FUNCTION_BLOCK FB_EVENT_LOGGER IMPLEMENTS I_EVENT_LOGGER
VAR
  fbAlarm:                        FB_TcAlarm;
  fbMessage:                      FB_TcMessage;
  bError:                         BOOL;
  bInfo:                          BOOL;
  bWarning:                       BOOL;
  uiSeq:                          ARRAY [1..3] OF UINT := [0, 0, 0];
  udiID:                          UDINT;
	sMsg:                           T_MaxString;
  bWithConfirmation:              BOOL;
END_VAR

IF bInfo THEN
  CASE uiSeq[1] OF
    0:
      fbMessage.CreateEx(TC_EVENTS.Info.IndividualInfoMsg, 0);
      uiSeq[1] := 1;
    1:
      fbMessage.ipArguments.Clear().AddDInt(udiID).AddString(sMsg);
      fbMessage.Send(0);
      uiSeq[1] := 2;
    2:
      bInfo := FALSE;
      uiSeq[1] := 0;
	END_CASE
END_IF

IF bWarning THEN
  CASE uiSeq[2] OF
    0:
      fbMessage.CreateEx(TC_EVENTS.Warnings.IndividualWarningMsg, 0);
      uiSeq[2] := 1;
    1:
      fbMessage.ipArguments.Clear().AddDInt(udiID).AddString(sMsg);
      fbMessage.Send(0);
      uiSeq[2] := 2;
    2:
      bWarning := FALSE;
      uiSeq[2] := 0;
	END_CASE
END_IF

IF bError THEN
  CASE uiSeq[3] OF
    0:
      fbAlarm.CreateEx(TC_EVENTS.Errors.IndividualErrMsg, bWithConfirmation, 0);
      uiSeq[3] := 1;
    1:
      fbAlarm.ipArguments.Clear().AddDInt(udiID).AddString(sMsg);
      fbAlarm.Raise(0);
      uiSeq[3] := 2;
    2:
      bError := FALSE;
      uiSeq[3] := 0;
	END_CASE
END_IF

METHOD M_ErrorMsg : BOOL
VAR_INPUT
	udiID:                        UDINT;
	sMsg:                         T_MaxString;
  bWithConfirmation:            BOOL;
END_VAR
M_ErrorMsg := THIS^.uiSeq[3] = 2;

// Assign input
THIS^.udiID := udiID;
THIS^.sMsg := sMsg;
THIS^.bWithConfirmation := bWithConfirmation;

THIS^.bError := TRUE;
END_METHOD

METHOD M_InfoMsg : BOOL
VAR_INPUT
	udiID	: UDINT;
	sMsg	: Tc2_System.T_MaxString;
END_VAR
M_InfoMsg := THIS^.uiSeq[1] = 2;

// Assign input
THIS^.udiID := udiID;
THIS^.sMsg := sMsg;

THIS^.bInfo := TRUE;
END_METHOD

{warning 'Methodenimplementierung hinzufügen'}
(*=== Method: M_Run  ============================================

 @brief: Here is the global code (Timer, Event, Flange,...)*)
METHOD M_Run
END_METHOD

METHOD M_WarningMsg : BOOL
VAR_INPUT
	udiID	: UDINT;
	sMsg	: Tc2_System.T_MaxString;
END_VAR
M_WarningMsg := THIS^.uiSeq[2] = 2;

// Assign input
THIS^.udiID := udiID;
THIS^.sMsg := sMsg;

THIS^.bWarning := TRUE;
END_METHOD

{warning 'Eigenschaftenimplementierung hinzufügen'}
(*=== Property: P_Event  ============================================

 @param [set]: 	Set the Structure "ST_EVENT" from another Object
 @param [get]: 	Return the Structure "ST_EVENT", it contains the actual 
					event of the Object *)
PROPERTY P_Event : GenLib.ST_EVENT
GET
END_GET
SET
END_SET
END_PROPERTY

{warning 'Eigenschaftenimplementierung hinzufügen'}
(*=== Property: P_FullObjectPath  ============================================

 @param [set]: 	Set the Object Path (Clear String of Object)
 @param [get]: 	Return the Objectpath *)
PROPERTY P_FullObjectPath : STRING
GET
END_GET
SET
END_SET
END_PROPERTY

{warning 'Eigenschaftenimplementierung hinzufügen'}
(*=== Property: P_Global_Ack  ============================================

 @param [set]: 	Set the Bit for Ack from another Object
 @param [get]: 	Return the state of Ack Bit*)
PROPERTY P_Global_Ack : BOOL
GET
END_GET
SET
END_SET
END_PROPERTY

{warning 'Eigenschaftenimplementierung hinzufügen'}
(*=== Property: P_GlobalID  ============================================

 @param [set]: 	-
 @param [get]: 	Return the string of instance path*)
PROPERTY P_GlobalID : STRING
GET
END_GET
END_PROPERTY

END_FUNCTION_BLOCK

(* stored: Version 1.1.0.1, ProductVersion 3.1.4024.12
   POU FB_EVENT_LOGGER: Id {c7a3cb00-eeb6-4905-8930-18e4802c682a}, SpecialFunc None
   Method M_ErrorMsg: Id {19fbce93-535e-4c73-b977-36e7db2a9ddb}
   Method M_InfoMsg: Id {fc354915-a515-4312-b3d4-f11cdd8da792}
   Method M_Run: Id {66457c75-ddcd-4157-b8bc-e20988a2f08e}
   Method M_WarningMsg: Id {b0dd5e76-edf9-46bb-bc0a-86e7f1896a38}
   Property P_Event: Id {771994c3-828a-4a10-a23b-b5fc6f7cd29b}
   Get Get: Id {f9827bf1-b722-4319-a974-50ebfd3b6ea5}
   Set Set: Id {ca3eae66-2ef2-40c3-ab81-03aba26cf8de}
   Property P_FullObjectPath: Id {caef1014-ae1f-4668-877b-a070794e9176}
   Get Get: Id {0b5e0e43-58de-4140-a23e-907d3efb380e}
   Set Set: Id {1e19d4b8-79b9-4739-bfb9-c58f09e3a121}
   Property P_Global_Ack: Id {34341a3f-3111-4f00-87d1-76b5271a51e1}
   Get Get: Id {82ceaebb-3f41-47b2-800a-51a6dbb04cc8}
   Set Set: Id {136551f6-2487-419e-9b98-ffb7bb105d4a}
   Property P_GlobalID: Id {5065b438-13ec-4f28-b43e-3f5a246524bc}
   Get Get: Id {cc53d8bb-4153-4ecf-8f58-30c70a036a14} *)
